(* IEC 61131-3 sources: elnaProjects/ElpcLogic/PomarKc7Changed/build_USO_ecl/_ (part 9) *)

FUNCTION nsCepeiControl : BOOL
  VAR_INPUT
    im : ImConfig;
  END_VAR

  nsCepeiControl:= NOT (
  	im.kran1.reliability OR
  	im.kran2.reliability OR
  	im.kran4.reliability OR
  	im.kran5.reliability OR
  	im.kran6.reliability OR
  	im.kran3b.reliability OR
  	im.pns.reliability OR
  	im.nu1.reliability OR
  	im.nu2.reliability OR
  	im.PNS.reliability OR
            im.v1_Avom.reliability OR
            im.v2_Avom.reliability OR
            (*im.Ten.reliability OR*)
  	im.mv.reliability);
END_FUNCTION

FUNCTION NapryageniaOK : BOOL
  VAR_INPUT
    im : ImConfig;
  END_VAR

  NapryageniaOK:=
  NOT (Im.SingleSignals.NS_G1_G2.Q
  OR Im.SingleSignals.NS_G10_G11.Q
  OR Im.SingleSignals.NS_G13_G14.Q
  OR Im.SingleSignals.NS_G15_G16.Q
  OR Im.SingleSignals.NS_G17.Q
  OR Im.SingleSignals.NS_G18_G19.Q
  OR Im.SingleSignals.NS_G3_G4.Q
  OR Im.SingleSignals.NS_G5_G6.Q
  OR Im.SingleSignals.NS_G7_G8.Q
  OR im.SingleSignals.QF1_on.Q
  OR Im.SingleSignals.QF2_on.Q
  OR Im.SingleSignals.QF23_on.Q
  OR Im.SingleSignals.QF4_QF5_on.Q
  OR Im.SingleSignals.QF6_QF7_on.Q
  OR Im.SingleSignals.QF8_QF9_on.Q
  OR Im.SingleSignals.QF10_QF11_on.Q
  OR im.SingleSignals.QF12_QF13_on.Q
  OR im.SingleSignals.QF22_on.Q
  OR Im.SingleSignals.QF14_QF15_on.Q);
END_FUNCTION

FUNCTION discretNS : BOOL
  VAR_INPUT
    di : DiConfig;
  END_VAR

  discretNS:=  ((di.di_0.reliability <> 255)
                OR (di.di_1.reliability <> 255)
                OR (di.di_2.reliability <> 255)
                OR (di.di_3.reliability <> 255)
                OR (di.di_4.reliability <> 255)
                OR (di.di_5.reliability <> 255)
                OR (di.di_6.reliability <> 255)
                OR (di.di_7.reliability <> 255)
                OR (di.di_8.reliability <> 255)
                OR (di.di_9.reliability <> 255)
                OR (di.di_10.reliability <> 255)
                OR (di.di_11.reliability <> 255)
                OR (di.di_12.reliability <> 255)
                OR (di.di_13.reliability <> 255)
                OR (di.di_14.reliability <> 255));
               (* OR (di.di_15.reliability <> 255)); *)
END_FUNCTION

FUNCTION BlockAllProtections : BOOL
  VAR_IN_OUT
    protections : ProtectionsConfig;
  END_VAR

  protections.Topornogo_podshipnika_EDT_1.inOpcCommandsDisabled:=TRUE;
  protections.Toy_podshipnika_EDT_2.inOpcCommandsDisabled:=TRUE;
  protections.Toy_podshipnika_kol_EDT_3.inOpcCommandsDisabled:=TRUE;
  protections.Toy_podshipnika_kol_EDT_4.inOpcCommandsDisabled:=TRUE;
  protections.To_podshipnika_shest_red_EDT_5.inOpcCommandsDisabled:=TRUE;
  protections.To_podshipnika_shest_red_EDT_6.inOpcCommandsDisabled:=TRUE;
  protections.To_podshipnika_N_EDT_7.inOpcCommandsDisabled:=TRUE;
  protections.To_podshipnika_svob_konca_EDT_8.inOpcCommandsDisabled:=TRUE;
  protections.Ty_podshipnika_rab_kol_EDT_9.inOpcCommandsDisabled:=TRUE;
  protections.Typornogo_podshipnika_nerab_kolodok_HT_10.inOpcCommandsDisabled:=TRUE;
  protections.Tgaza_na_vyhode_H.inOpcCommandsDisabled:=TRUE;
  protections.Os_sdvig_nagnetatelja_plus.inOpcCommandsDisabled:=TRUE;
  protections.Os_sdvig_nagnetatelja_minus.inOpcCommandsDisabled:=TRUE;
  protections.Pgaza_na_vyhode_nagnetatelia_GPA_STOP.inOpcCommandsDisabled:=TRUE;
  protections.Pgaza_na_vhode_nagnetatelia_GPA_STOP.inOpcCommandsDisabled:=TRUE;
  protections.Pgaza_na_vyhode_nagnetatelia.inOpcCommandsDisabled:=TRUE;
  protections.dPmaslo_gaz.inOpcCommandsDisabled:=TRUE;
  protections.Pmaslo_sm_nizkoe.inOpcCommandsDisabled:=TRUE;
  protections.Pmaslo_sm_vysokoe.inOpcCommandsDisabled:=TRUE;
  protections.Vibro_skorost_OPED_T1.inOpcCommandsDisabled:=TRUE;
  protections.Vibro_skorost_OPED_T2.inOpcCommandsDisabled:=TRUE;
  protections.Vibro_skorost_OYP_kolesa_ED_T3.inOpcCommandsDisabled:=TRUE;
  protections.Vibro_skorost_OP_kolesa_RH_T4.inOpcCommandsDisabled:=TRUE;
  protections.Vibro_skorost_OP_shesterni_RED_T5.inOpcCommandsDisabled:=TRUE;
  protections.Vibro_skorost_OP_shesterni_RED_T6.inOpcCommandsDisabled:=TRUE;
  protections.dPmaslo_gaz_less100.inOpcCommandsDisabled:=TRUE;
  protections.Reg_vozb_off.inOpcCommandsDisabled:=TRUE;
  protections.Fail_chastotnii_pusk.inOpcCommandsDisabled:=TRUE;
  protections.Off_avar_vikluchatel.inOpcCommandsDisabled:=TRUE;
  protections.AOKC_SHKC.inOpcCommandsDisabled:=TRUE;
  protections.AO_PRU.inOpcCommandsDisabled:=TRUE;
  protections.AO_ot_SHU.inOpcCommandsDisabled:=TRUE;
  protections.mvOff.inOpcCommandsDisabled:=TRUE;
  protections.Kran1_sdvig.inOpcCommandsDisabled:=TRUE;
  protections.Kran2_sdvig.inOpcCommandsDisabled:=TRUE;
END_FUNCTION

PROGRAM program0
  VAR
    SysTime : LREAL;
    systime_ns : ULINT;
    systime_s : ULINT;
    preSysTime : LREAL;
    tmpCycle : LREAL;
    preSys_s : ULINT;
    preSys_ns : ULINT;
  END_VAR
  VAR_EXTERNAL
    cur_Cycle : REAL;
    gStart_Tmr : REAL;
  END_VAR
  VAR
    Timings : fb_Timings;
    _init : BOOL      := TRUE;
    life_count : UINT;
    AI_structs_ini : proc_AI_Init;
    AI_Proc : proc_AI;
    AO_structs_ini : proc_AO_Init;
    AO_Proc : proc_AO;
    DI_structs_ini : proc_DI_Init;
    DI_Proc : proc_DI;
    DO_structs_ini : proc_DO_Init;
    DO_Proc : proc_DO;
    Get_algoritms_OPC : OPC_algoritms_set;
    Set_algoritms_OPC : OPC_algoritms_get;
    IM_structs_ini : proc_IM_Init;
    IM_Proc : proc_IM;
    Protections_structs_ini : proc_Protections_Init;
    Protections_Proc : proc_Protection;
    Algoritms_Proc : proc_algoritms;
    AlgoritmsManager : fb_AlgoritmsManager;
    ProtectionsManager : fb_ProtectionsManager;
  END_VAR
  VAR_EXTERNAL
    algManager : struct_AlgoritmsManager;
    protectManager : struct_ProtectionsManager;
  END_VAR

  (* Обработка времени. *)
  SysTime := ULINT_TO_LREAL(systime_s) + (1.0E-9 * ULINT_TO_LREAL(systime_ns));
  preSysTime := SysTime;
  tmpCycle := ULINT_TO_LREAL(systime_s - preSys_s) + 1.0E-9 * (ULINT_TO_LREAL(systime_ns) - ULINT_TO_LREAL(preSys_ns));
  cur_Cycle := LREAL_TO_REAL(tmpCycle);
  preSys_s := systime_s;
  preSys_ns := systime_ns;
  IF gStart_Tmr < 99999.9 THEN gStart_Tmr := gStart_Tmr + cur_Cycle; END_IF;
  Timings();

  IF  _init (*or external_init_ai *) then           (* Требуется инициализация структур и ФБ. *)
    (* Инициализация аналоговых входов. *)
      AI_structs_ini(init := TRUE);
      AI_Proc((*init := FALSE*));

    (* Инициализация дискретных входов. *)
      DI_structs_ini(init := TRUE);
      DI_Proc((*init := FALSE*));

      (* Инициализация аналоговых выходов. *)
  (*     AO_structs_ini(init := TRUE);
         AO_Proc(init := TRUE);*)

    (* Инициализация дискретных выходов. *)
      DO_structs_ini(init := TRUE);
      DO_Proc((*init := FALSE*));

     (* Инициализация ИМ. *)
      IM_structs_ini(init := TRUE);
      IM_Proc();

     (* Инициализация Защит *)
      Protections_structs_ini(init := TRUE);
      (*Protections_Proc();*)

       (* Стартовая инициализация OPC-тэгов элементами канальных структур. *)
          (*___________________AI______________________________________________________________________________*)
      (*ini_AI_OPC();*)

      _init := FALSE;

    ELSE                         (* Завершена инициализация структур и ФБ. *)

  (* Перенос OPC-тэгов в элементы структур каналов. *)
        (*___________________________________________AI________________________________________________*)
      (*Get_AI_OPC(); *)
       Get_algoritms_OPC();

     (* Пересчёт защит САУ. *)
     ProtectionsManager(protectManager);

       (* Пересчёт алгоритмов САУ. *)
     AlgoritmsManager(algManager);

      (****               Опрос входов.              ****)
          (* Опрос аналоговых входов. *)
      AI_Proc((*init := FALSE*));

          (* Опрос дискретных входов. *)
      DI_Proc((*init := FALSE*));

      (****              Запись выходов.             ****)
          (* Запись аналоговых выходов. *)
  (*    AO_Proc(init := FALSE);*)

       (* Запись дискретных выходов. *)
      DO_Proc((*init := FALSE*));

      (****               Опрос ИМ              ****)
      IM_Proc();

      (****            Опрос Защит              ****)
      Protections_Proc();

      Algoritms_Proc();

  END_IF;

  (* Передача информации на верхний уровень по OPC UA протоколу. *)
    (* Передача состояний каналов AI. *)
  (*Set_AI_OPC();)*
  (* Передача состояний каналов ИМ. *)
  (* Передача состояний защит. *)
  (* Передача состояний алгоритмов. *)
  Set_algoritms_OPC();
END_PROGRAM

CONFIGURATION config1
  VAR_GLOBAL
    systime_s AT %IL0.10.10 : ULINT;
    systime_ns AT %IL0.10.11 : ULINT;
    current_retrieve_us AT %IL0.10.12 : ULINT;
    current_config_us AT %IL0.10.13 : ULINT;
    current_publish_us AT %IL0.10.14 : ULINT;
    current_run_us AT %IL0.10.15 : ULINT;
    max_retrieve_us AT %QL0.10.16 : ULINT;
    max_config_us AT %QL0.10.17 : ULINT;
    max_publish_us AT %QL0.10.18 : ULINT;
    plc_run_number AT %IL0.10.19 : ULINT;
    arAIN_0 : TItemAIN;
    arAIN_1 : TItemAIN;
    arAIN_2 : TItemAIN;
    arAIN_3 : TItemAIN;
    arAIN_4 : TItemAIN;
    arAIN_5 : TItemAIN;
    arAIN_6 : TItemAIN;
    arAIN_7 : TItemAIN;
    arAIN_8 : TItemAIN;
    arAIN_9 : TItemAIN;
    arAIN_10 : TItemAIN;
    arAIN_11 : TItemAIN;
    arAIN_12 : TItemAIN;
    arAIN_13 : TItemAIN;
    arAIN_14 : TItemAIN;
    arAIN_15 : TItemAIN;
    arAIN_16 : TItemAIN;
    arAIN_17 : TItemAIN;
    arAIN_18 : TItemAIN;
    arAIN_19 : TItemAIN;
    arAIN_20 : TItemAIN;
    arAIN_21 : TItemAIN;
    arAIN_22 : TItemAIN;
    arAIN_23 : TItemAIN;
    arAIN_24 : TItemAIN;
    arAIN_25 : TItemAIN;
    arAIN_26 : TItemAIN;
    arAIN_27 : TItemAIN;
    arAIN_28 : TItemAIN;
    arAIN_29 : TItemAIN;
    arAIN_30 : TItemAIN;
    arAIN_31 : TItemAIN;
    arAIN_32 : TItemAIN;
    arAIN_33 : TItemAIN;
    arAIN_34 : TItemAIN;
    arAIN_35 : TItemAIN;
    arAIN_36 : TItemAIN;
    arAIN_37 : TItemAIN;
    arAIN_38 : TItemAIN;
    arAIN_39 : TItemAIN;
    arAIN_40 : TItemAIN;
    arAIN_41 : TItemAIN;
    arAIN_42 : TItemAIN;
    arAIN_43 : TItemAIN;
    arAIN_44 : TItemAIN;
    arAIN_45 : TItemAIN;
    arAIN_46 : TItemAIN;
    arAIN_47 : TItemAIN;
    arAIN_48 : TItemAIN;
    arAIN_49 : TItemAIN;
    arAIN_50 : TItemAIN;
    arAIN_51 : TItemAIN;
    arAIN_52 : TItemAIN;
    arAIN_53 : TItemAIN;
    arAIN_54 : TItemAIN;
    arAIN_55 : TItemAIN;
    arAIN_56 : TItemAIN;
    arAIN_57 : TItemAIN;
    arAIN_58 : TItemAIN;
    arAIN_59 : TItemAIN;
    arAIN_60 : TItemAIN;
    arAIN_61 : TItemAIN;
    arAIN_62 : TItemAIN;
    arAIN_63 : TItemAIN;
    arAIN_64 : TItemAIN;
    arAIN_65 : TItemAIN;
    arAIN_66 : TItemAIN;
    arAIN_67 : TItemAIN;
    arAIN_68 : TItemAIN;
    arAIN_69 : TItemAIN;
    arAIN_70 : TItemAIN;
    arAIN_71 : TItemAIN;
    arAIN_72 : TItemAIN;
    arAIN_73 : TItemAIN;
    arAIN_74 : TItemAIN;
    arAIN_75 : TItemAIN;
    arAIN_76 : TItemAIN;
    arAIN_77 : TItemAIN;
    arAIN_78 : TItemAIN;
    arAIN_79 : TItemAIN;
    arDIN_0 : TItemDIN;
    arDIN_1 : TItemDIN;
    arDIN_2 : TItemDIN;
    arDIN_3 : TItemDIN;
    arDIN_4 : TItemDIN;
    arDIN_5 : TItemDIN;
    arDIN_6 : TItemDIN;
    arDIN_7 : TItemDIN;
    arDIN_8 : TItemDIN;
    arDIN_9 : TItemDIN;
    arDIN_10 : TItemDIN;
    arDIN_11 : TItemDIN;
    arDIN_12 : TItemDIN;
    arDIN_13 : TItemDIN;
    arDIN_14 : TItemDIN;
    arDIN_15 : TItemDIN;
    arDIN_16 : TItemDIN;
    arDIN_17 : TItemDIN;
    arDIN_18 : TItemDIN;
    arDIN_19 : TItemDIN;
    arDIN_20 : TItemDIN;
    arDIN_21 : TItemDIN;
    arAOUT_0 : TDoubleData;
    arAOUT_1 : TDoubleData;
    arDOUT_0 : TWordData;
    arDOUT_1 : TWordData;
    arDOUT_2 : TWordData;
    arDOUT_3 : TWordData;
    arDOUT_4 : TWordData;
    arDOUT_66 : TWordData;
    arERR_0 : TItemDIN;
    arERR_1 : TItemDIN;
    arERR_2 : TItemDIN;
    arERR_3 : TItemDIN;
    arERR_4 : TItemDIN;
    arERR_5 : TItemDIN;
    arERR_6 : TItemDIN;
    arERR_7 : TItemDIN;
    arERR_8 : TItemDIN;
    arERR_9 : TItemDIN;
    arERR_10 : TItemDIN;
    arERR_11 : TItemDIN;
    arERR_12 : TItemDIN;
    arERR_13 : TItemDIN;
    arERR_14 : TItemDIN;
    arERR_15 : TItemDIN;
    arERR_16 : TItemDIN;
    arERR_17 : TItemDIN;
    arERR_18 : TItemDIN;
    arERR_19 : TItemDIN;
    arERR_20 : TItemDIN;
    arERR_21 : TItemDIN;
    arERR_22 : TItemDIN;
    arERR_23 : TItemDIN;
    arERR_24 : TItemDIN;
    arERR_66 : TItemDIN;
    arRelSt_0 : TItemDIN;
  END_VAR

  RESOURCE resource1 ON PLC
    VAR_GLOBAL CONSTANT
      gMaint_Time : REAL;
    END_VAR
    VAR_GLOBAL
      cur_Cycle : REAL;
      gStart_Tmr : REAL;
    END_VAR
    VAR_GLOBAL CONSTANT
      req_Cycle : REAL := 0.02;
    END_VAR
    VAR_GLOBAL
      gF_T_100mSec : BOOL;
      gT_1Sec : BOOL;
      gF_T_1Sec : BOOL;
      gT_1Min : BOOL;
      gR_T_1Min : BOOL;
      gF_T_1Min : BOOL;
      T_1SEC : REAL;
      del_T : REAL;
      ai : AiConfig;
      di : DiConfig;
      od : DOconfig;
      ao : AOConfig;
      IM : ImConfig;
      protections : ProtectionsConfig;
      algoritms : AlgoritmsConfig;
      algManager : struct_AlgoritmsManager;
      ModeGpa : TYPE_ModeGpa;
      protectManager : struct_ProtectionsManager;
      NotHasRezervNU : BOOL;
      Reset_HasNU : BOOL;
      AlgTimers : struct_AlgTimers;
      AlgQuestions : AlgoritmsQuestions;
      PMcommand : TYPE_CommandsPotectionsManager;
      AI_Aktivnaia_moshchnost_HL AT %QL0.2 : LREAL;
      AI_Aktivnaia_moshchnost_LL AT %QL0.3 : LREAL;
      AI_Aktivnaia_moshchnost_command AT %QW0.1 : UINT;
      AI_Aktivnaia_moshchnost_newHL AT %QL0.4 : LREAL;
      AI_Aktivnaia_moshchnost_newLL AT %QL0.5 : LREAL;
      AI_Aktivnaia_moshchnost_status AT %QD0.6 : UDINT;
      AI_Aktivnaia_moshchnost_value AT %QL0.7 : LREAL;
      AI_Osevoi_sdvig_rotora_nagnetatelia_HA AT %QL0.27 : LREAL;
      AI_Osevoi_sdvig_rotora_nagnetatelia_HL AT %QL0.28 : LREAL;
      AI_Osevoi_sdvig_rotora_nagnetatelia_HW AT %QL0.29 : LREAL;
      AI_Osevoi_sdvig_rotora_nagnetatelia_LA AT %QL0.30 : LREAL;
      AI_Osevoi_sdvig_rotora_nagnetatelia_LL AT %QL0.31 : LREAL;
      AI_Osevoi_sdvig_rotora_nagnetatelia_LW AT %QL0.32 : LREAL;
      AI_Osevoi_sdvig_rotora_nagnetatelia_command AT %QW0.26 : UINT;
      AI_Osevoi_sdvig_rotora_nagnetatelia_newHA AT %QL0.33 : LREAL;
      AI_Osevoi_sdvig_rotora_nagnetatelia_newHL AT %QL0.34 : LREAL;
      AI_Osevoi_sdvig_rotora_nagnetatelia_newHW AT %QL0.35 : LREAL;
      AI_Osevoi_sdvig_rotora_nagnetatelia_newLA AT %QL0.36 : LREAL;
      AI_Osevoi_sdvig_rotora_nagnetatelia_newLL AT %QL0.37 : LREAL;
      AI_Osevoi_sdvig_rotora_nagnetatelia_newLW AT %QL0.38 : LREAL;
      AI_Osevoi_sdvig_rotora_nagnetatelia_status AT %QD0.39 : UDINT;
      AI_Osevoi_sdvig_rotora_nagnetatelia_value AT %QL0.40 : LREAL;
      AI_P_gaza_na_vkhode_nagnetatelia_HL AT %QL0.42 : LREAL;
      AI_P_gaza_na_vkhode_nagnetatelia_LL AT %QL0.43 : LREAL;
      AI_P_gaza_na_vkhode_nagnetatelia_command AT %QW0.41 : UINT;
      AI_P_gaza_na_vkhode_nagnetatelia_newHL AT %QL0.44 : LREAL;
      AI_P_gaza_na_vkhode_nagnetatelia_newLL AT %QL0.45 : LREAL;
      AI_P_gaza_na_vkhode_nagnetatelia_status AT %QD0.46 : UDINT;
      AI_P_gaza_na_vkhode_nagnetatelia_value AT %QL0.47 : LREAL;
      AI_P_gaza_na_vykhode_nagnetatelia_HL AT %QL0.49 : LREAL;
      AI_P_gaza_na_vykhode_nagnetatelia_LL AT %QL0.50 : LREAL;
      AI_P_gaza_na_vykhode_nagnetatelia_command AT %QW0.48 : UINT;
      AI_P_gaza_na_vykhode_nagnetatelia_newHL AT %QL0.51 : LREAL;
      AI_P_gaza_na_vykhode_nagnetatelia_newLL AT %QL0.52 : LREAL;
      AI_P_gaza_na_vykhode_nagnetatelia_status AT %QD0.53 : UDINT;
      AI_P_gaza_na_vykhode_nagnetatelia_value AT %QL0.54 : LREAL;
      AI_P_masla_smazki_nizkoe_HL AT %QL0.56 : LREAL;
      AI_P_masla_smazki_nizkoe_LA AT %QL0.57 : LREAL;
      AI_P_masla_smazki_nizkoe_LL AT %QL0.58 : LREAL;
      AI_P_masla_smazki_nizkoe_LW AT %QL0.59 : LREAL;
      AI_P_masla_smazki_nizkoe_command AT %QW0.55 : UINT;
      AI_P_masla_smazki_nizkoe_newHL AT %QL0.60 : LREAL;
      AI_P_masla_smazki_nizkoe_newLA AT %QL0.61 : LREAL;
      AI_P_masla_smazki_nizkoe_newLL AT %QL0.62 : LREAL;
      AI_P_masla_smazki_nizkoe_newLW AT %QL0.63 : LREAL;
      AI_P_masla_smazki_nizkoe_status AT %QD0.64 : UDINT;
      AI_P_masla_smazki_nizkoe_value AT %QL0.65 : LREAL;
      AI_P_masla_smazki_srednee_posle_nasosov_HL AT %QL0.67 : LREAL;
      AI_P_masla_smazki_srednee_posle_nasosov_LL AT %QL0.68 : LREAL;
      AI_P_masla_smazki_srednee_posle_nasosov_LW AT %QL0.69 : LREAL;
      AI_P_masla_smazki_srednee_posle_nasosov_command AT %QW0.66 : UINT;
      AI_P_masla_smazki_srednee_posle_nasosov_newHL AT %QL0.70 : LREAL;
      AI_P_masla_smazki_srednee_posle_nasosov_newLL AT %QL0.71 : LREAL;
      AI_P_masla_smazki_srednee_posle_nasosov_newLW AT %QL0.72 : LREAL;
      AI_P_masla_smazki_srednee_posle_nasosov_status AT %QD0.73 : UDINT;
      AI_P_masla_smazki_srednee_posle_nasosov_value AT %QL0.74 : LREAL;
      AI_P_masla_uplotneniia_HL AT %QL0.76 : LREAL;
      AI_P_masla_uplotneniia_LL AT %QL0.77 : LREAL;
      AI_P_masla_uplotneniia_command AT %QW0.75 : UINT;
      AI_P_masla_uplotneniia_newHL AT %QL0.78 : LREAL;
      AI_P_masla_uplotneniia_newLL AT %QL0.79 : LREAL;
      AI_P_masla_uplotneniia_status AT %QD0.80 : UDINT;
      AI_P_masla_uplotneniia_value AT %QL0.81 : LREAL;
      AI_Reaktivnaia_moshchnost_HL AT %QL0.83 : LREAL;
      AI_Reaktivnaia_moshchnost_LL AT %QL0.84 : LREAL;
      AI_Reaktivnaia_moshchnost_command AT %QW0.82 : UINT;
      AI_Reaktivnaia_moshchnost_newHL AT %QL0.85 : LREAL;
      AI_Reaktivnaia_moshchnost_newLL AT %QL0.86 : LREAL;
      AI_Reaktivnaia_moshchnost_status AT %QD0.87 : UDINT;
      AI_Reaktivnaia_moshchnost_value AT %QL0.88 : LREAL;
      AI_T_aktivnogo_zheleza_statora_1_k_HL AT %QL0.90 : LREAL;
      AI_T_aktivnogo_zheleza_statora_1_k_LL AT %QL0.91 : LREAL;
      AI_T_aktivnogo_zheleza_statora_1_k_command AT %QW0.89 : UINT;
      AI_T_aktivnogo_zheleza_statora_1_k_newHL AT %QL0.92 : LREAL;
      AI_T_aktivnogo_zheleza_statora_1_k_newLL AT %QL0.93 : LREAL;
      AI_T_aktivnogo_zheleza_statora_1_k_status AT %QD0.94 : UDINT;
      AI_T_aktivnogo_zheleza_statora_1_k_value AT %QL0.95 : LREAL;
      AI_T_aktivnogo_zheleza_statora_2_k_HL AT %QL0.97 : LREAL;
      AI_T_aktivnogo_zheleza_statora_2_k_LL AT %QL0.98 : LREAL;
      AI_T_aktivnogo_zheleza_statora_2_k_command AT %QW0.96 : UINT;
      AI_T_aktivnogo_zheleza_statora_2_k_newHL AT %QL0.99 : LREAL;
      AI_T_aktivnogo_zheleza_statora_2_k_newLL AT %QL0.100 : LREAL;
      AI_T_aktivnogo_zheleza_statora_2_k_status AT %QD0.101 : UDINT;
      AI_T_aktivnogo_zheleza_statora_2_k_value AT %QL0.102 : LREAL;
      AI_T_aktivnogo_zheleza_statora_3_k_HL AT %QL0.104 : LREAL;
      AI_T_aktivnogo_zheleza_statora_3_k_LL AT %QL0.105 : LREAL;
      AI_T_aktivnogo_zheleza_statora_3_k_command AT %QW0.103 : UINT;
      AI_T_aktivnogo_zheleza_statora_3_k_newHL AT %QL0.106 : LREAL;
      AI_T_aktivnogo_zheleza_statora_3_k_newLL AT %QL0.107 : LREAL;
      AI_T_aktivnogo_zheleza_statora_3_k_status AT %QD0.108 : UDINT;
      AI_T_aktivnogo_zheleza_statora_3_k_value AT %QL0.109 : LREAL;
      AI_T_clodAir_dvigatelia_t1_HL AT %QL0.111 : LREAL;
      AI_T_clodAir_dvigatelia_t1_LL AT %QL0.112 : LREAL;
      AI_T_clodAir_dvigatelia_t1_command AT %QW0.110 : UINT;
      AI_T_clodAir_dvigatelia_t1_newHL AT %QL0.113 : LREAL;
      AI_T_clodAir_dvigatelia_t1_newLL AT %QL0.114 : LREAL;
      AI_T_clodAir_dvigatelia_t1_status AT %QD0.115 : UDINT;
      AI_T_clodAir_dvigatelia_t1_value AT %QL0.116 : LREAL;
      AI_T_gaz_in_nagnetatelia_HL AT %QL0.118 : LREAL;
      AI_T_gaz_in_nagnetatelia_LL AT %QL0.119 : LREAL;
      AI_T_gaz_in_nagnetatelia_command AT %QW0.117 : UINT;
      AI_T_gaz_in_nagnetatelia_newHL AT %QL0.120 : LREAL;
      AI_T_gaz_in_nagnetatelia_newLL AT %QL0.121 : LREAL;
      AI_T_gaz_in_nagnetatelia_status AT %QD0.122 : UDINT;
      AI_T_gaz_in_nagnetatelia_value AT %QL0.123 : LREAL;
      AI_T_gaz_out_nagnetatelia_HA AT %QL0.125 : LREAL;
      AI_T_gaz_out_nagnetatelia_HL AT %QL0.126 : LREAL;
      AI_T_gaz_out_nagnetatelia_HW AT %QL0.127 : LREAL;
      AI_T_gaz_out_nagnetatelia_LL AT %QL0.128 : LREAL;
      AI_T_gaz_out_nagnetatelia_command AT %QW0.124 : UINT;
      AI_T_gaz_out_nagnetatelia_newHA AT %QL0.129 : LREAL;
      AI_T_gaz_out_nagnetatelia_newHL AT %QL0.130 : LREAL;
      AI_T_gaz_out_nagnetatelia_newHW AT %QL0.131 : LREAL;
      AI_T_gaz_out_nagnetatelia_newLL AT %QL0.132 : LREAL;
      AI_T_gaz_out_nagnetatelia_status AT %QD0.133 : UDINT;
      AI_T_gaz_out_nagnetatelia_value AT %QL0.134 : LREAL;
      AI_T_hotAir_dvigatelia_t1_HL AT %QL0.136 : LREAL;
      AI_T_hotAir_dvigatelia_t1_LL AT %QL0.137 : LREAL;
      AI_T_hotAir_dvigatelia_t1_command AT %QW0.135 : UINT;
      AI_T_hotAir_dvigatelia_t1_newHL AT %QL0.138 : LREAL;
      AI_T_hotAir_dvigatelia_t1_newLL AT %QL0.139 : LREAL;
      AI_T_hotAir_dvigatelia_t1_status AT %QD0.140 : UDINT;
      AI_T_hotAir_dvigatelia_t1_value AT %QL0.141 : LREAL;
      AI_T_masla_do_AVOM_HL AT %QL0.143 : LREAL;
      AI_T_masla_do_AVOM_LL AT %QL0.144 : LREAL;
      AI_T_masla_do_AVOM_command AT %QW0.142 : UINT;
      AI_T_masla_do_AVOM_newHL AT %QL0.145 : LREAL;
      AI_T_masla_do_AVOM_newLL AT %QL0.146 : LREAL;
      AI_T_masla_do_AVOM_status AT %QD0.147 : UDINT;
      AI_T_masla_do_AVOM_value AT %QL0.148 : LREAL;
      AI_T_masla_na_slive_perednego_opornogo_podshipnika_dvigatelia_HL AT %QL0.150 : LREAL;
      AI_T_masla_na_slive_perednego_opornogo_podshipnika_dvigatelia_LL AT %QL0.151 : LREAL;
      AI_T_masla_na_slive_perednego_opornogo_podshipnika_dvigatelia_command AT %QW0.149 : UINT;
      AI_T_masla_na_slive_perednego_opornogo_podshipnika_dvigatelia_newHL AT %QL0.152 : LREAL;
      AI_T_masla_na_slive_perednego_opornogo_podshipnika_dvigatelia_newLL AT %QL0.153 : LREAL;
      AI_T_masla_na_slive_perednego_opornogo_podshipnika_dvigatelia_status AT %QD0.154 : UDINT;
      AI_T_masla_na_slive_perednego_opornogo_podshipnika_dvigatelia_value AT %QL0.155 : LREAL;
      AI_T_masla_na_slive_zadnego_opornogo_podshipnika_dvigatelia_HL AT %QL0.157 : LREAL;
      AI_T_masla_na_slive_zadnego_opornogo_podshipnika_dvigatelia_LL AT %QL0.158 : LREAL;
      AI_T_masla_na_slive_zadnego_opornogo_podshipnika_dvigatelia_command AT %QW0.156 : UINT;
      AI_T_masla_na_slive_zadnego_opornogo_podshipnika_dvigatelia_newHL AT %QL0.159 : LREAL;
      AI_T_masla_na_slive_zadnego_opornogo_podshipnika_dvigatelia_newLL AT %QL0.160 : LREAL;
      AI_T_masla_na_slive_zadnego_opornogo_podshipnika_dvigatelia_status AT %QD0.161 : UDINT;
      AI_T_masla_na_slive_zadnego_opornogo_podshipnika_dvigatelia_value AT %QL0.162 : LREAL;
      AI_T_masla_posle_AVOM_HL AT %QL0.164 : LREAL;
      AI_T_masla_posle_AVOM_LL AT %QL0.165 : LREAL;
      AI_T_masla_posle_AVOM_command AT %QW0.163 : UINT;
      AI_T_masla_posle_AVOM_newHL AT %QL0.166 : LREAL;
      AI_T_masla_posle_AVOM_newLL AT %QL0.167 : LREAL;
      AI_T_masla_posle_AVOM_status AT %QD0.168 : UDINT;
      AI_T_masla_posle_AVOM_value AT %QL0.169 : LREAL;
      AI_T_masla_v_maslobake_HL AT %QL0.171 : LREAL;
      AI_T_masla_v_maslobake_HW AT %QL0.172 : LREAL;
      AI_T_masla_v_maslobake_LL AT %QL0.173 : LREAL;
      AI_T_masla_v_maslobake_LW AT %QL0.174 : LREAL;
      AI_T_masla_v_maslobake_command AT %QW0.170 : UINT;
      AI_T_masla_v_maslobake_newHL AT %QL0.175 : LREAL;
      AI_T_masla_v_maslobake_newHW AT %QL0.176 : LREAL;
      AI_T_masla_v_maslobake_newLL AT %QL0.177 : LREAL;
      AI_T_masla_v_maslobake_newLW AT %QL0.178 : LREAL;
      AI_T_masla_v_maslobake_status AT %QD0.179 : UDINT;
      AI_T_masla_v_maslobake_value AT %QL0.180 : LREAL;
      AI_T_obmotki_fazy_1_k_HL AT %QL0.182 : LREAL;
      AI_T_obmotki_fazy_1_k_LL AT %QL0.183 : LREAL;
      AI_T_obmotki_fazy_1_k_command AT %QW0.181 : UINT;
      AI_T_obmotki_fazy_1_k_newHL AT %QL0.184 : LREAL;
      AI_T_obmotki_fazy_1_k_newLL AT %QL0.185 : LREAL;
      AI_T_obmotki_fazy_1_k_status AT %QD0.186 : UDINT;
      AI_T_obmotki_fazy_1_k_value AT %QL0.187 : LREAL;
      AI_T_obmotki_fazy_2_k_HL AT %QL0.189 : LREAL;
      AI_T_obmotki_fazy_2_k_LL AT %QL0.190 : LREAL;
      AI_T_obmotki_fazy_2_k_command AT %QW0.188 : UINT;
      AI_T_obmotki_fazy_2_k_newHL AT %QL0.191 : LREAL;
      AI_T_obmotki_fazy_2_k_newLL AT %QL0.192 : LREAL;
      AI_T_obmotki_fazy_2_k_status AT %QD0.193 : UDINT;
      AI_T_obmotki_fazy_2_k_value AT %QL0.194 : LREAL;
      AI_T_obmotki_fazy_3_k_HL AT %QL0.196 : LREAL;
      AI_T_obmotki_fazy_3_k_LL AT %QL0.197 : LREAL;
      AI_T_obmotki_fazy_3_k_command AT %QW0.195 : UINT;
      AI_T_obmotki_fazy_3_k_newHL AT %QL0.198 : LREAL;
      AI_T_obmotki_fazy_3_k_newLL AT %QL0.199 : LREAL;
      AI_T_obmotki_fazy_3_k_status AT %QD0.200 : UDINT;
      AI_T_obmotki_fazy_3_k_value AT %QL0.201 : LREAL;
      AI_T_oporno_upornogo_podshipnika_nagnetatelia_t4_HA AT %QL0.203 : LREAL;
      AI_T_oporno_upornogo_podshipnika_nagnetatelia_t4_HL AT %QL0.204 : LREAL;
      AI_T_oporno_upornogo_podshipnika_nagnetatelia_t4_HW AT %QL0.205 : LREAL;
      AI_T_oporno_upornogo_podshipnika_nagnetatelia_t4_LL AT %QL0.206 : LREAL;
      AI_T_oporno_upornogo_podshipnika_nagnetatelia_t4_command AT %QW0.202 : UINT;
      AI_T_oporno_upornogo_podshipnika_nagnetatelia_t4_newHA AT %QL0.207 : LREAL;
      AI_T_oporno_upornogo_podshipnika_nagnetatelia_t4_newHL AT %QL0.208 : LREAL;
      AI_T_oporno_upornogo_podshipnika_nagnetatelia_t4_newHW AT %QL0.209 : LREAL;
      AI_T_oporno_upornogo_podshipnika_nagnetatelia_t4_newLL AT %QL0.210 : LREAL;
      AI_T_oporno_upornogo_podshipnika_nagnetatelia_t4_status AT %QD0.211 : UDINT;
      AI_T_oporno_upornogo_podshipnika_nagnetatelia_t4_value AT %QL0.212 : LREAL;
      AI_T_opornogo_podshipnika_nagnetatelia_t1_HA AT %QL0.214 : LREAL;
      AI_T_opornogo_podshipnika_nagnetatelia_t1_HL AT %QL0.215 : LREAL;
      AI_T_opornogo_podshipnika_nagnetatelia_t1_HW AT %QL0.216 : LREAL;
      AI_T_opornogo_podshipnika_nagnetatelia_t1_LL AT %QL0.217 : LREAL;
      AI_T_opornogo_podshipnika_nagnetatelia_t1_command AT %QW0.213 : UINT;
      AI_T_opornogo_podshipnika_nagnetatelia_t1_newHA AT %QL0.218 : LREAL;
      AI_T_opornogo_podshipnika_nagnetatelia_t1_newHL AT %QL0.219 : LREAL;
      AI_T_opornogo_podshipnika_nagnetatelia_t1_newHW AT %QL0.220 : LREAL;
      AI_T_opornogo_podshipnika_nagnetatelia_t1_newLL AT %QL0.221 : LREAL;
      AI_T_opornogo_podshipnika_nagnetatelia_t1_status AT %QD0.222 : UDINT;
      AI_T_opornogo_podshipnika_nagnetatelia_t1_value AT %QL0.223 : LREAL;
      AI_T_opornogo_podshipnika_nagnetatelia_t2_HA AT %QL0.225 : LREAL;
      AI_T_opornogo_podshipnika_nagnetatelia_t2_HL AT %QL0.226 : LREAL;
      AI_T_opornogo_podshipnika_nagnetatelia_t2_HW AT %QL0.227 : LREAL;
      AI_T_opornogo_podshipnika_nagnetatelia_t2_LL AT %QL0.228 : LREAL;
      AI_T_opornogo_podshipnika_nagnetatelia_t2_command AT %QW0.224 : UINT;
      AI_T_opornogo_podshipnika_nagnetatelia_t2_newHA AT %QL0.229 : LREAL;
      AI_T_opornogo_podshipnika_nagnetatelia_t2_newHL AT %QL0.230 : LREAL;
      AI_T_opornogo_podshipnika_nagnetatelia_t2_newHW AT %QL0.231 : LREAL;
      AI_T_opornogo_podshipnika_nagnetatelia_t2_newLL AT %QL0.232 : LREAL;
      AI_T_opornogo_podshipnika_nagnetatelia_t2_status AT %QD0.233 : UDINT;
      AI_T_opornogo_podshipnika_nagnetatelia_t2_value AT %QL0.234 : LREAL;
      AI_T_opornogo_podshipnika_nagnetatelia_t3_HA AT %QL0.236 : LREAL;
      AI_T_opornogo_podshipnika_nagnetatelia_t3_HL AT %QL0.237 : LREAL;
      AI_T_opornogo_podshipnika_nagnetatelia_t3_HW AT %QL0.238 : LREAL;
      AI_T_opornogo_podshipnika_nagnetatelia_t3_LL AT %QL0.239 : LREAL;
      AI_T_opornogo_podshipnika_nagnetatelia_t3_command AT %QW0.235 : UINT;
      AI_T_opornogo_podshipnika_nagnetatelia_t3_newHA AT %QL0.240 : LREAL;
      AI_T_opornogo_podshipnika_nagnetatelia_t3_newHL AT %QL0.241 : LREAL;
      AI_T_opornogo_podshipnika_nagnetatelia_t3_newHW AT %QL0.242 : LREAL;
      AI_T_opornogo_podshipnika_nagnetatelia_t3_newLL AT %QL0.243 : LREAL;
      AI_T_opornogo_podshipnika_nagnetatelia_t3_status AT %QD0.244 : UDINT;
      AI_T_opornogo_podshipnika_nagnetatelia_t3_value AT %QL0.245 : LREAL;
      AI_T_perednego_opornogo_podshipnika_dvigatelia_t1_HA AT %QL0.247 : LREAL;
      AI_T_perednego_opornogo_podshipnika_dvigatelia_t1_HL AT %QL0.248 : LREAL;
      AI_T_perednego_opornogo_podshipnika_dvigatelia_t1_HW AT %QL0.249 : LREAL;
      AI_T_perednego_opornogo_podshipnika_dvigatelia_t1_LL AT %QL0.250 : LREAL;
      AI_T_perednego_opornogo_podshipnika_dvigatelia_t1_command AT %QW0.246 : UINT;
      AI_T_perednego_opornogo_podshipnika_dvigatelia_t1_newHA AT %QL0.251 : LREAL;
      AI_T_perednego_opornogo_podshipnika_dvigatelia_t1_newHL AT %QL0.252 : LREAL;
      AI_T_perednego_opornogo_podshipnika_dvigatelia_t1_newHW AT %QL0.253 : LREAL;
      AI_T_perednego_opornogo_podshipnika_dvigatelia_t1_newLL AT %QL0.254 : LREAL;
      AI_T_perednego_opornogo_podshipnika_dvigatelia_t1_status AT %QD0.255 : UDINT;
      AI_T_perednego_opornogo_podshipnika_dvigatelia_t1_value AT %QL0.256 : LREAL;
      AI_T_podshipnika_reduktora_t1_HA AT %QL0.258 : LREAL;
      AI_T_podshipnika_reduktora_t1_HL AT %QL0.259 : LREAL;
      AI_T_podshipnika_reduktora_t1_HW AT %QL0.260 : LREAL;
      AI_T_podshipnika_reduktora_t1_LL AT %QL0.261 : LREAL;
      AI_T_podshipnika_reduktora_t1_command AT %QW0.257 : UINT;
      AI_T_podshipnika_reduktora_t1_newHA AT %QL0.262 : LREAL;
      AI_T_podshipnika_reduktora_t1_newHL AT %QL0.263 : LREAL;
      AI_T_podshipnika_reduktora_t1_newHW AT %QL0.264 : LREAL;
      AI_T_podshipnika_reduktora_t1_newLL AT %QL0.265 : LREAL;
      AI_T_podshipnika_reduktora_t1_status AT %QD0.266 : UDINT;
      AI_T_podshipnika_reduktora_t1_value AT %QL0.267 : LREAL;
      AI_T_podshipnika_reduktora_t2_HA AT %QL0.269 : LREAL;
      AI_T_podshipnika_reduktora_t2_HL AT %QL0.270 : LREAL;
      AI_T_podshipnika_reduktora_t2_HW AT %QL0.271 : LREAL;
      AI_T_podshipnika_reduktora_t2_LL AT %QL0.272 : LREAL;
      AI_T_podshipnika_reduktora_t2_command AT %QW0.268 : UINT;
      AI_T_podshipnika_reduktora_t2_newHA AT %QL0.273 : LREAL;
      AI_T_podshipnika_reduktora_t2_newHL AT %QL0.274 : LREAL;
      AI_T_podshipnika_reduktora_t2_newHW AT %QL0.275 : LREAL;
      AI_T_podshipnika_reduktora_t2_newLL AT %QL0.276 : LREAL;
      AI_T_podshipnika_reduktora_t2_status AT %QD0.277 : UDINT;
      AI_T_podshipnika_reduktora_t2_value AT %QL0.278 : LREAL;
      AI_T_podshipnika_reduktora_t3_HA AT %QL0.280 : LREAL;
      AI_T_podshipnika_reduktora_t3_HL AT %QL0.281 : LREAL;
      AI_T_podshipnika_reduktora_t3_HW AT %QL0.282 : LREAL;
      AI_T_podshipnika_reduktora_t3_LL AT %QL0.283 : LREAL;
      AI_T_podshipnika_reduktora_t3_command AT %QW0.279 : UINT;
      AI_T_podshipnika_reduktora_t3_newHA AT %QL0.284 : LREAL;
      AI_T_podshipnika_reduktora_t3_newHL AT %QL0.285 : LREAL;
      AI_T_podshipnika_reduktora_t3_newHW AT %QL0.286 : LREAL;
      AI_T_podshipnika_reduktora_t3_newLL AT %QL0.287 : LREAL;
      AI_T_podshipnika_reduktora_t3_status AT %QD0.288 : UDINT;
      AI_T_podshipnika_reduktora_t3_value AT %QL0.289 : LREAL;
      AI_T_podshipnika_reduktora_t4_HA AT %QL0.291 : LREAL;
      AI_T_podshipnika_reduktora_t4_HL AT %QL0.292 : LREAL;
      AI_T_podshipnika_reduktora_t4_HW AT %QL0.293 : LREAL;
      AI_T_podshipnika_reduktora_t4_LL AT %QL0.294 : LREAL;
      AI_T_podshipnika_reduktora_t4_command AT %QW0.290 : UINT;
      AI_T_podshipnika_reduktora_t4_newHA AT %QL0.295 : LREAL;
      AI_T_podshipnika_reduktora_t4_newHL AT %QL0.296 : LREAL;
      AI_T_podshipnika_reduktora_t4_newHW AT %QL0.297 : LREAL;
      AI_T_podshipnika_reduktora_t4_newLL AT %QL0.298 : LREAL;
      AI_T_podshipnika_reduktora_t4_status AT %QD0.299 : UDINT;
      AI_T_podshipnika_reduktora_t4_value AT %QL0.300 : LREAL;
      AI_T_vnytri_shkafa_HL AT %QL0.866 : LREAL;
      AI_T_vnytri_shkafa_HW AT %QL0.870 : LREAL;
      AI_T_vnytri_shkafa_LL AT %QL0.867 : LREAL;
      AI_T_vnytri_shkafa_LW AT %QL0.872 : LREAL;
      AI_T_vnytri_shkafa_command AT %QW0.863 : UINT;
      AI_T_vnytri_shkafa_newHL AT %QL0.868 : LREAL;
      AI_T_vnytri_shkafa_newHW AT %QL0.871 : LREAL;
      AI_T_vnytri_shkafa_newLL AT %QL0.869 : LREAL;
      AI_T_vnytri_shkafa_newLW AT %QL0.873 : LREAL;
      AI_T_vnytri_shkafa_status AT %QD0.864 : UDINT;
      AI_T_vnytri_shkafa_value AT %QL0.865 : LREAL;
      AI_T_zadnego_opornogo_podshipnika_dvigatelia_t2_HA AT %QL0.302 : LREAL;
      AI_T_zadnego_opornogo_podshipnika_dvigatelia_t2_HL AT %QL0.303 : LREAL;
      AI_T_zadnego_opornogo_podshipnika_dvigatelia_t2_HW AT %QL0.304 : LREAL;
      AI_T_zadnego_opornogo_podshipnika_dvigatelia_t2_LL AT %QL0.305 : LREAL;
      AI_T_zadnego_opornogo_podshipnika_dvigatelia_t2_command AT %QW0.301 : UINT;
      AI_T_zadnego_opornogo_podshipnika_dvigatelia_t2_newHA AT %QL0.306 : LREAL;
      AI_T_zadnego_opornogo_podshipnika_dvigatelia_t2_newHL AT %QL0.307 : LREAL;
      AI_T_zadnego_opornogo_podshipnika_dvigatelia_t2_newHW AT %QL0.308 : LREAL;
      AI_T_zadnego_opornogo_podshipnika_dvigatelia_t2_newLL AT %QL0.309 : LREAL;
      AI_T_zadnego_opornogo_podshipnika_dvigatelia_t2_status AT %QD0.310 : UDINT;
      AI_T_zadnego_opornogo_podshipnika_dvigatelia_t2_value AT %QL0.311 : LREAL;
      AI_Tok_statora_elektrodvigatelia_HL AT %QL0.313 : LREAL;
      AI_Tok_statora_elektrodvigatelia_LL AT %QL0.314 : LREAL;
      AI_Tok_statora_elektrodvigatelia_command AT %QW0.312 : UINT;
      AI_Tok_statora_elektrodvigatelia_newHL AT %QL0.315 : LREAL;
      AI_Tok_statora_elektrodvigatelia_newLL AT %QL0.316 : LREAL;
      AI_Tok_statora_elektrodvigatelia_status AT %QD0.317 : UDINT;
      AI_Tok_statora_elektrodvigatelia_value AT %QL0.318 : LREAL;
      AI_Tok_vozbuzhdeniia_vozbuditelia_HL AT %QL0.320 : LREAL;
      AI_Tok_vozbuzhdeniia_vozbuditelia_LL AT %QL0.321 : LREAL;
      AI_Tok_vozbuzhdeniia_vozbuditelia_command AT %QW0.319 : UINT;
      AI_Tok_vozbuzhdeniia_vozbuditelia_newHL AT %QL0.322 : LREAL;
      AI_Tok_vozbuzhdeniia_vozbuditelia_newLL AT %QL0.323 : LREAL;
      AI_Tok_vozbuzhdeniia_vozbuditelia_status AT %QD0.324 : UDINT;
      AI_Tok_vozbuzhdeniia_vozbuditelia_value AT %QL0.325 : LREAL;
      AI_Uroven_masla_v_maslobake_HL AT %QL0.327 : LREAL;
      AI_Uroven_masla_v_maslobake_HW AT %QL0.328 : LREAL;
      AI_Uroven_masla_v_maslobake_LA AT %QL0.329 : LREAL;
      AI_Uroven_masla_v_maslobake_LL AT %QL0.330 : LREAL;
      AI_Uroven_masla_v_maslobake_LW AT %QL0.331 : LREAL;
      AI_Uroven_masla_v_maslobake_command AT %QW0.326 : UINT;
      AI_Uroven_masla_v_maslobake_newHL AT %QL0.332 : LREAL;
      AI_Uroven_masla_v_maslobake_newHW AT %QL0.333 : LREAL;
      AI_Uroven_masla_v_maslobake_newLA AT %QL0.334 : LREAL;
      AI_Uroven_masla_v_maslobake_newLL AT %QL0.335 : LREAL;
      AI_Uroven_masla_v_maslobake_newLW AT %QL0.336 : LREAL;
      AI_Uroven_masla_v_maslobake_status AT %QD0.337 : UDINT;
      AI_Uroven_masla_v_maslobake_value AT %QL0.338 : LREAL;
      AI_Vibratciia_STD_t1_HA AT %QL0.384 : LREAL;
      AI_Vibratciia_STD_t1_HL AT %QL0.385 : LREAL;
      AI_Vibratciia_STD_t1_HW AT %QL0.386 : LREAL;
      AI_Vibratciia_STD_t1_LL AT %QL0.387 : LREAL;
      AI_Vibratciia_STD_t1_command AT %QW0.383 : UINT;
      AI_Vibratciia_STD_t1_newHA AT %QL0.388 : LREAL;
      AI_Vibratciia_STD_t1_newHL AT %QL0.389 : LREAL;
      AI_Vibratciia_STD_t1_newHW AT %QL0.390 : LREAL;
      AI_Vibratciia_STD_t1_newLL AT %QL0.391 : LREAL;
      AI_Vibratciia_STD_t1_status AT %QD0.392 : UDINT;
      AI_Vibratciia_STD_t1_value AT %QL0.393 : LREAL;
      AI_Vibratciia_STD_t2_HA AT %QL0.395 : LREAL;
      AI_Vibratciia_STD_t2_HL AT %QL0.396 : LREAL;
      AI_Vibratciia_STD_t2_HW AT %QL0.397 : LREAL;
      AI_Vibratciia_STD_t2_LL AT %QL0.398 : LREAL;
      AI_Vibratciia_STD_t2_command AT %QW0.394 : UINT;
      AI_Vibratciia_STD_t2_newHA AT %QL0.399 : LREAL;
      AI_Vibratciia_STD_t2_newHL AT %QL0.400 : LREAL;
      AI_Vibratciia_STD_t2_newHW AT %QL0.401 : LREAL;
      AI_Vibratciia_STD_t2_newLL AT %QL0.402 : LREAL;
      AI_Vibratciia_STD_t2_status AT %QD0.403 : UDINT;
      AI_Vibratciia_STD_t2_value AT %QL0.404 : LREAL;
      AI_Vibratciia_rotora_nagnetatelia_t1_HA AT %QL0.340 : LREAL;
      AI_Vibratciia_rotora_nagnetatelia_t1_HL AT %QL0.341 : LREAL;
      AI_Vibratciia_rotora_nagnetatelia_t1_HW AT %QL0.342 : LREAL;
      AI_Vibratciia_rotora_nagnetatelia_t1_LL AT %QL0.343 : LREAL;
      AI_Vibratciia_rotora_nagnetatelia_t1_command AT %QW0.339 : UINT;
      AI_Vibratciia_rotora_nagnetatelia_t1_newHA AT %QL0.344 : LREAL;
      AI_Vibratciia_rotora_nagnetatelia_t1_newHL AT %QL0.345 : LREAL;
      AI_Vibratciia_rotora_nagnetatelia_t1_newHW AT %QL0.346 : LREAL;
      AI_Vibratciia_rotora_nagnetatelia_t1_newLL AT %QL0.347 : LREAL;
      AI_Vibratciia_rotora_nagnetatelia_t1_status AT %QD0.348 : UDINT;
      AI_Vibratciia_rotora_nagnetatelia_t1_value AT %QL0.349 : LREAL;
      AI_Vibratciia_rotora_nagnetatelia_t2_HA AT %QL0.351 : LREAL;
      AI_Vibratciia_rotora_nagnetatelia_t2_HL AT %QL0.352 : LREAL;
      AI_Vibratciia_rotora_nagnetatelia_t2_HW AT %QL0.353 : LREAL;
      AI_Vibratciia_rotora_nagnetatelia_t2_LL AT %QL0.354 : LREAL;
      AI_Vibratciia_rotora_nagnetatelia_t2_command AT %QW0.350 : UINT;
      AI_Vibratciia_rotora_nagnetatelia_t2_newHA AT %QL0.355 : LREAL;
      AI_Vibratciia_rotora_nagnetatelia_t2_newHL AT %QL0.356 : LREAL;
      AI_Vibratciia_rotora_nagnetatelia_t2_newHW AT %QL0.357 : LREAL;
      AI_Vibratciia_rotora_nagnetatelia_t2_newLL AT %QL0.358 : LREAL;
      AI_Vibratciia_rotora_nagnetatelia_t2_status AT %QD0.359 : UDINT;
      AI_Vibratciia_rotora_nagnetatelia_t2_value AT %QL0.360 : LREAL;
      AI_Vibratciia_rotora_nagnetatelia_t3_HA AT %QL0.362 : LREAL;
      AI_Vibratciia_rotora_nagnetatelia_t3_HL AT %QL0.363 : LREAL;
      AI_Vibratciia_rotora_nagnetatelia_t3_HW AT %QL0.364 : LREAL;
      AI_Vibratciia_rotora_nagnetatelia_t3_LL AT %QL0.365 : LREAL;
      AI_Vibratciia_rotora_nagnetatelia_t3_command AT %QW0.361 : UINT;
      AI_Vibratciia_rotora_nagnetatelia_t3_newHA AT %QL0.366 : LREAL;
      AI_Vibratciia_rotora_nagnetatelia_t3_newHL AT %QL0.367 : LREAL;
      AI_Vibratciia_rotora_nagnetatelia_t3_newHW AT %QL0.368 : LREAL;
      AI_Vibratciia_rotora_nagnetatelia_t3_newLL AT %QL0.369 : LREAL;
      AI_Vibratciia_rotora_nagnetatelia_t3_status AT %QD0.370 : UDINT;
      AI_Vibratciia_rotora_nagnetatelia_t3_value AT %QL0.371 : LREAL;
      AI_Vibratciia_rotora_nagnetatelia_t4_HA AT %QL0.373 : LREAL;
      AI_Vibratciia_rotora_nagnetatelia_t4_HL AT %QL0.374 : LREAL;
      AI_Vibratciia_rotora_nagnetatelia_t4_HW AT %QL0.375 : LREAL;
      AI_Vibratciia_rotora_nagnetatelia_t4_LL AT %QL0.376 : LREAL;
      AI_Vibratciia_rotora_nagnetatelia_t4_command AT %QW0.372 : UINT;
      AI_Vibratciia_rotora_nagnetatelia_t4_newHA AT %QL0.377 : LREAL;
      AI_Vibratciia_rotora_nagnetatelia_t4_newHL AT %QL0.378 : LREAL;
      AI_Vibratciia_rotora_nagnetatelia_t4_newHW AT %QL0.379 : LREAL;
      AI_Vibratciia_rotora_nagnetatelia_t4_newLL AT %QL0.380 : LREAL;
      AI_Vibratciia_rotora_nagnetatelia_t4_status AT %QD0.381 : UDINT;
      AI_Vibratciia_rotora_nagnetatelia_t4_value AT %QL0.382 : LREAL;
      AI_VoltageSHU_osnovnoi_vvod_HL AT %QL0.406 : LREAL;
      AI_VoltageSHU_osnovnoi_vvod_HW AT %QL0.407 : LREAL;
      AI_VoltageSHU_osnovnoi_vvod_LL AT %QL0.408 : LREAL;
      AI_VoltageSHU_osnovnoi_vvod_LW AT %QL0.409 : LREAL;
      AI_VoltageSHU_osnovnoi_vvod_command AT %QW0.405 : UINT;
      AI_VoltageSHU_osnovnoi_vvod_newHL AT %QL0.410 : LREAL;
      AI_VoltageSHU_osnovnoi_vvod_newHW AT %QL0.411 : LREAL;
      AI_VoltageSHU_osnovnoi_vvod_newLL AT %QL0.412 : LREAL;
      AI_VoltageSHU_osnovnoi_vvod_newLW AT %QL0.413 : LREAL;
      AI_VoltageSHU_osnovnoi_vvod_status AT %QD0.414 : UDINT;
      AI_VoltageSHU_osnovnoi_vvod_value AT %QL0.415 : LREAL;
      AI_VoltageSHU_rezervnyi_vvod_HL AT %QL0.417 : LREAL;
      AI_VoltageSHU_rezervnyi_vvod_HW AT %QL0.418 : LREAL;
      AI_VoltageSHU_rezervnyi_vvod_LL AT %QL0.419 : LREAL;
      AI_VoltageSHU_rezervnyi_vvod_LW AT %QL0.420 : LREAL;
      AI_VoltageSHU_rezervnyi_vvod_command AT %QW0.416 : UINT;
      AI_VoltageSHU_rezervnyi_vvod_newHL AT %QL0.421 : LREAL;
      AI_VoltageSHU_rezervnyi_vvod_newHW AT %QL0.422 : LREAL;
      AI_VoltageSHU_rezervnyi_vvod_newLL AT %QL0.423 : LREAL;
      AI_VoltageSHU_rezervnyi_vvod_newLW AT %QL0.424 : LREAL;
      AI_VoltageSHU_rezervnyi_vvod_status AT %QD0.425 : UDINT;
      AI_VoltageSHU_rezervnyi_vvod_value AT %QL0.426 : LREAL;
      AI_dP_gaza_na_konfuzore_nagnetatelia_HL AT %QL0.9 : LREAL;
      AI_dP_gaza_na_konfuzore_nagnetatelia_LL AT %QL0.10 : LREAL;
      AI_dP_gaza_na_konfuzore_nagnetatelia_command AT %QW0.8 : UINT;
      AI_dP_gaza_na_konfuzore_nagnetatelia_newHL AT %QL0.11 : LREAL;
      AI_dP_gaza_na_konfuzore_nagnetatelia_newLL AT %QL0.12 : LREAL;
      AI_dP_gaza_na_konfuzore_nagnetatelia_status AT %QD0.13 : UDINT;
      AI_dP_gaza_na_konfuzore_nagnetatelia_value AT %QL0.14 : LREAL;
      AI_dPmaslo_gaz_HL AT %QL0.16 : LREAL;
      AI_dPmaslo_gaz_LA AT %QL0.17 : LREAL;
      AI_dPmaslo_gaz_LL AT %QL0.18 : LREAL;
      AI_dPmaslo_gaz_LW AT %QL0.19 : LREAL;
      AI_dPmaslo_gaz_MaxChangeDown AT %QL0.877 : LREAL;
      AI_dPmaslo_gaz_MaxChangeUP AT %QL0.876 : LREAL;
      AI_dPmaslo_gaz_command AT %QW0.15 : UINT;
      AI_dPmaslo_gaz_newHL AT %QL0.20 : LREAL;
      AI_dPmaslo_gaz_newLA AT %QL0.21 : LREAL;
      AI_dPmaslo_gaz_newLL AT %QL0.22 : LREAL;
      AI_dPmaslo_gaz_newLW AT %QL0.23 : LREAL;
      AI_dPmaslo_gaz_newMaxChangeDown AT %QL0.875 : LREAL;
      AI_dPmaslo_gaz_newMaxChangeUP AT %QL0.874 : LREAL;
      AI_dPmaslo_gaz_status AT %QD0.24 : UDINT;
      AI_dPmaslo_gaz_value AT %QL0.25 : LREAL;
      A1_10_err_mode AT %QW0.825 : UINT;
      A1_11_err_mode AT %QW0.826 : UINT;
      A1_12_err_mode AT %QW0.827 : UINT;
      A1_13_err_mode AT %QW0.828 : UINT;
      A1_14_err_mode AT %QW0.829 : UINT;
      A1_15_err_mode AT %QW0.830 : UINT;
      A1_1_err_mode AT %QW0.816 : UINT;
      A1_2_err_mode AT %QW0.817 : UINT;
      A1_3_err_mode AT %QW0.818 : UINT;
      A1_4_err_mode AT %QW0.819 : UINT;
      A1_5_err_mode AT %QW0.820 : UINT;
      A1_6_err_mode AT %QW0.821 : UINT;
      A1_7_err_mode AT %QW0.822 : UINT;
      A1_8_err_mode AT %QW0.823 : UINT;
      A1_9_err_mode AT %QW0.824 : UINT;
      A2_10_err_mode AT %QW0.840 : UINT;
      A2_11_err_mode AT %QW0.841 : UINT;
      A2_12_err_mode AT %QW0.842 : UINT;
      A2_13_err_mode AT %QW0.843 : UINT;
      A2_14_err_mode AT %QW0.844 : UINT;
      A2_15_err_mode AT %QW0.845 : UINT;
      A2_1_err_mode AT %QW0.831 : UINT;
      A2_2_err_mode AT %QW0.832 : UINT;
      A2_3_err_mode AT %QW0.833 : UINT;
      A2_4_err_mode AT %QW0.834 : UINT;
      A2_5_err_mode AT %QW0.835 : UINT;
      A2_6_err_mode AT %QW0.836 : UINT;
      A2_7_err_mode AT %QW0.837 : UINT;
      A2_8_err_mode AT %QW0.838 : UINT;
      A2_9_err_mode AT %QW0.839 : UINT;
      AI_0_dblValue AT %QL0.736 : LREAL;
      AI_10_dblValue AT %QL0.746 : LREAL;
      AI_11_dblValue AT %QL0.747 : LREAL;
      AI_12_dblValue AT %QL0.748 : LREAL;
      AI_13_dblValue AT %QL0.749 : LREAL;
      AI_14_dblValue AT %QL0.750 : LREAL;
      AI_15_dblValue AT %QL0.751 : LREAL;
      AI_16_dblValue AT %QL0.752 : LREAL;
      AI_17_dblValue AT %QL0.753 : LREAL;
      AI_18_dblValue AT %QL0.754 : LREAL;
      AI_19_dblValue AT %QL0.755 : LREAL;
      AI_1_dblValue AT %QL0.737 : LREAL;
      AI_20_dblValue AT %QL0.756 : LREAL;
      AI_21_dblValue AT %QL0.757 : LREAL;
      AI_22_dblValue AT %QL0.758 : LREAL;
      AI_23_dblValue AT %QL0.759 : LREAL;
      AI_24_dblValue AT %QL0.760 : LREAL;
      AI_25_dblValue AT %QL0.761 : LREAL;
      AI_26_dblValue AT %QL0.762 : LREAL;
      AI_27_dblValue AT %QL0.763 : LREAL;
      AI_28_dblValue AT %QL0.764 : LREAL;
      AI_29_dblValue AT %QL0.765 : LREAL;
      AI_2_dblValue AT %QL0.738 : LREAL;
      AI_30_dblValue AT %QL0.766 : LREAL;
      AI_31_dblValue AT %QL0.767 : LREAL;
      AI_32_dblValue AT %QL0.768 : LREAL;
      AI_33_dblValue AT %QL0.769 : LREAL;
      AI_34_dblValue AT %QL0.770 : LREAL;
      AI_35_dblValue AT %QL0.771 : LREAL;
      AI_36_dblValue AT %QL0.772 : LREAL;
      AI_37_dblValue AT %QL0.773 : LREAL;
      AI_38_dblValue AT %QL0.774 : LREAL;
      AI_39_dblValue AT %QL0.775 : LREAL;
      AI_3_dblValue AT %QL0.739 : LREAL;
      AI_40_dblValue AT %QL0.776 : LREAL;
      AI_41_dblValue AT %QL0.777 : LREAL;
      AI_42_dblValue AT %QL0.778 : LREAL;
      AI_43_dblValue AT %QL0.779 : LREAL;
      AI_44_dblValue AT %QL0.780 : LREAL;
      AI_45_dblValue AT %QL0.781 : LREAL;
      AI_46_dblValue AT %QL0.782 : LREAL;
      AI_47_dblValue AT %QL0.783 : LREAL;
      AI_48_dblValue AT %QL0.784 : LREAL;
      AI_49_dblValue AT %QL0.785 : LREAL;
      AI_4_dblValue AT %QL0.740 : LREAL;
      AI_50_dblValue AT %QL0.786 : LREAL;
      AI_51_dblValue AT %QL0.787 : LREAL;
      AI_52_dblValue AT %QL0.788 : LREAL;
      AI_53_dblValue AT %QL0.789 : LREAL;
      AI_54_dblValue AT %QL0.790 : LREAL;
      AI_55_dblValue AT %QL0.791 : LREAL;
      AI_56_dblValue AT %QL0.792 : LREAL;
      AI_57_dblValue AT %QL0.793 : LREAL;
      AI_58_dblValue AT %QL0.794 : LREAL;
      AI_59_dblValue AT %QL0.795 : LREAL;
      AI_5_dblValue AT %QL0.741 : LREAL;
      AI_60_dblValue AT %QL0.796 : LREAL;
      AI_61_dblValue AT %QL0.797 : LREAL;
      AI_62_dblValue AT %QL0.798 : LREAL;
      AI_63_dblValue AT %QL0.799 : LREAL;
      AI_64_dblValue AT %QL0.800 : LREAL;
      AI_65_dblValue AT %QL0.801 : LREAL;
      AI_66_dblValue AT %QL0.802 : LREAL;
      AI_67_dblValue AT %QL0.803 : LREAL;
      AI_68_dblValue AT %QL0.804 : LREAL;
      AI_69_dblValue AT %QL0.805 : LREAL;
      AI_6_dblValue AT %QL0.742 : LREAL;
      AI_70_dblValue AT %QL0.806 : LREAL;
      AI_71_dblValue AT %QL0.807 : LREAL;
      AI_72_dblValue AT %QL0.808 : LREAL;
      AI_73_dblValue AT %QL0.809 : LREAL;
      AI_74_dblValue AT %QL0.810 : LREAL;
      AI_75_dblValue AT %QL0.811 : LREAL;
      AI_76_dblValue AT %QL0.812 : LREAL;
      AI_77_dblValue AT %QL0.813 : LREAL;
      AI_78_dblValue AT %QL0.814 : LREAL;
      AI_79_dblValue AT %QL0.815 : LREAL;
      AI_7_dblValue AT %QL0.743 : LREAL;
      AI_8_dblValue AT %QL0.744 : LREAL;
      AI_9_dblValue AT %QL0.745 : LREAL;
      BS_Core1 AT %QD0.603 : REAL;
      BS_Core2 AT %QD0.675 : REAL;
      BS_Core3 AT %QD0.683 : REAL;
      BS_Core4 AT %QD0.709 : REAL;
      BS_FreeMemory AT %QD0.730 : REAL;
      BS_Temp1 AT %QD0.734 : REAL;
      BS_Temp2 AT %QD0.735 : REAL;
      DI_0_1_wValue AT %QD0.852 : UDINT;
      DI_10_11_wValue AT %QD0.857 : UDINT;
      DI_12_13_wValue AT %QD0.858 : UDINT;
      DI_14_15_wValue AT %QD0.859 : UDINT;
      DI_16_17_wValue AT %QD0.860 : UDINT;
      DI_18_19_wValue AT %QD0.861 : UDINT;
      DI_20_21_wValue AT %QD0.862 : UDINT;
      DI_2_3_wValue AT %QD0.853 : UDINT;
      DI_4_5_wValue AT %QD0.854 : UDINT;
      DI_6_7_wValue AT %QD0.855 : UDINT;
      DI_8_9_wValue AT %QD0.856 : UDINT;
      DO_0_wValue AT %QW0.846 : UINT;
      DO_1_wValue AT %QW0.847 : UINT;
      DO_2_wValue AT %QW0.848 : UINT;
      DO_3_wValue AT %QW0.849 : UINT;
      DO_4_wValue AT %QW0.850 : UINT;
      DO_5_wValue AT %QW0.851 : UINT;
      IM_SingleSignals_DverShkafaOtkryta_status AT %QD0.456 : UDINT;
      IM_SingleSignals_KZ_10kv_status AT %QD0.457 : UDINT;
      IM_SingleSignals_NOGPA_knopkaSHU_status AT %QD0.453 : UDINT;
      IM_SingleSignals_NS_G10_G11_status AT %QD0.481 : UDINT;
      IM_SingleSignals_NS_G13_G14_status AT %QD0.482 : UDINT;
      IM_SingleSignals_NS_G15_G16_status AT %QD0.483 : UDINT;
      IM_SingleSignals_NS_G17_status AT %QD0.484 : UDINT;
      IM_SingleSignals_NS_G18_G19_status AT %QD0.485 : UDINT;
      IM_SingleSignals_NS_G1_G2_status AT %QD0.477 : UDINT;
      IM_SingleSignals_NS_G3_G4_status AT %QD0.478 : UDINT;
      IM_SingleSignals_NS_G5_G6_status AT %QD0.479 : UDINT;
      IM_SingleSignals_NS_G7_G8_status AT %QD0.480 : UDINT;
      IM_SingleSignals_OsevoiSdvig_levo_status AT %QD0.458 : UDINT;
      IM_SingleSignals_OsevoiSdvig_pravo_status AT %QD0.459 : UDINT;
      IM_SingleSignals_P_oil_low_status AT %QD0.455 : UDINT;
      IM_SingleSignals_QF10_QF11_on_status AT %QD0.463 : UDINT;
      IM_SingleSignals_QF12_QF13_on_status AT %QD0.464 : UDINT;
      IM_SingleSignals_QF14_QF15_on_status AT %QD0.465 : UDINT;
      IM_SingleSignals_QF1_on_status AT %QD0.466 : UDINT;
      IM_SingleSignals_QF22_on_status AT %QD0.476 : UDINT;
      IM_SingleSignals_QF23_on_status AT %QD0.468 : UDINT;
      IM_SingleSignals_QF2_on_status AT %QD0.467 : UDINT;
      IM_SingleSignals_QF4_QF5_on_status AT %QD0.460 : UDINT;
      IM_SingleSignals_QF6_QF7_on_status AT %QD0.461 : UDINT;
      IM_SingleSignals_QF8_QF9_on_status AT %QD0.462 : UDINT;
      IM_SingleSignals_Vozb_AsinchHod_status AT %QD0.469 : UDINT;
      IM_SingleSignals_Vozb_ControlVozbuditela_status AT %QD0.470 : UDINT;
      IM_SingleSignals_Vozb_KontaktorON_status AT %QD0.471 : UDINT;
      IM_SingleSignals_Vozb_Overload_status AT %QD0.472 : UDINT;
      IM_SingleSignals_Vozb_ProboiVentila_status AT %QD0.473 : UDINT;
      IM_SingleSignals_Vozb_ReSynchronize_status AT %QD0.474 : UDINT;
      IM_SingleSignals_dP_gazgaz_Kran1_status AT %QD0.454 : UDINT;
      IM_SingleSignals_dP_oilgaz_low_status AT %QD0.475 : UDINT;
      IM_Ten_inCommand_ARM AT %QW0.447 : UINT;
      IM_Ten_status AT %QD0.448 : UDINT;
      IM_kran1_inCommand_ARM AT %QW0.427 : UINT;
      IM_kran1_status AT %QD0.428 : UDINT;
      IM_kran2_inCommand_ARM AT %QW0.429 : UINT;
      IM_kran2_status AT %QD0.430 : UDINT;
      IM_kran3b_inCommand_ARM AT %QW0.431 : UINT;
      IM_kran3b_status AT %QD0.432 : UDINT;
      IM_kran4_inCommand_ARM AT %QW0.433 : UINT;
      IM_kran4_status AT %QD0.434 : UDINT;
      IM_kran5_inCommand_ARM AT %QW0.435 : UINT;
      IM_kran5_status AT %QD0.436 : UDINT;
      IM_kran6_inCommand_ARM AT %QW0.437 : UINT;
      IM_kran6_status AT %QD0.438 : UDINT;
      IM_mv_inCommand_ARM AT %QW0.439 : UINT;
      IM_mv_status AT %QD0.440 : UDINT;
      IM_nu1_inCommand_ARM AT %QW0.441 : UINT;
      IM_nu1_status AT %QD0.442 : UDINT;
      IM_nu2_inCommand_ARM AT %QW0.443 : UINT;
      IM_nu2_status AT %QD0.444 : UDINT;
      IM_pns_inCommand_ARM AT %QW0.445 : UINT;
      IM_pns_status AT %QD0.446 : UDINT;
      IM_v1_Avom_inCommand_ARM AT %QW0.449 : UINT;
      IM_v1_Avom_status AT %QD0.450 : UDINT;
      IM_v2_Avom_inCommand_ARM AT %QW0.451 : UINT;
      IM_v2_Avom_status AT %QD0.452 : UDINT;
      algManager_Mode AT %QW0.732 : UINT;
      algoritms_AntiPompag_UgolVNA_Value AT %QL0.726 : LREAL;
      algoritms_AntiPompag_UgolVNA_inCommand_ARM AT %QW0.605 : UINT;
      algoritms_AntiPompag_UgolVNA_newValue AT %QL0.606 : LREAL;
      algoritms_AntiPompag_UgolVNA_status AT %QD0.725 : UDINT;
      algoritms_AntiPompag_q_Value AT %QL0.724 : LREAL;
      algoritms_AntiPompag_q_inCommand_ARM AT %QW0.604 : UINT;
      algoritms_AntiPompag_q_status AT %QD0.723 : UDINT;
      algoritms_AntiPompag_zapas_Value AT %QL0.728 : LREAL;
      algoritms_AntiPompag_zapas_inCommand_ARM AT %QW0.607 : UINT;
      algoritms_AntiPompag_zapas_status AT %QD0.727 : UDINT;
      algoritms_Apusk_Error AT %QD0.689 : UDINT;
      algoritms_Apusk_Start AT %QD0.688 : UDINT;
      algoritms_Apusk_Top AT %QD0.690 : UDINT;
      algoritms_Apusk_inCommand_ARM AT %QW0.555 : UINT;
      algoritms_Apusk_status AT %QD0.687 : UDINT;
      algoritms_AutoAvom_hysteresis_Value AT %QL0.716 : LREAL;
      algoritms_AutoAvom_hysteresis_inCommand_ARM AT %QW0.556 : UINT;
      algoritms_AutoAvom_hysteresis_newValue AT %QL0.557 : LREAL;
      algoritms_AutoAvom_hysteresis_status AT %QD0.715 : UDINT;
      algoritms_AutoAvom_inCommand_ARM AT %QW0.562 : UINT;
      algoritms_AutoAvom_on1Temperature_Value AT %QL0.712 : LREAL;
      algoritms_AutoAvom_on1Temperature_inCommand_ARM AT %QW0.558 : UINT;
      algoritms_AutoAvom_on1Temperature_newValue AT %QL0.559 : LREAL;
      algoritms_AutoAvom_on1Temperature_status AT %QD0.711 : UDINT;
      algoritms_AutoAvom_on2Temperature_Value AT %QL0.714 : LREAL;
      algoritms_AutoAvom_on2Temperature_inCommand_ARM AT %QW0.560 : UINT;
      algoritms_AutoAvom_on2Temperature_newValue AT %QL0.561 : LREAL;
      algoritms_AutoAvom_on2Temperature_status AT %QD0.713 : UDINT;
      algoritms_AutoAvom_status AT %QD0.710 : UDINT;
      algoritms_AutoPns_OffTimer AT %QW0.701 : UINT;
      algoritms_AutoPns_OnTimer AT %QW0.700 : UINT;
      algoritms_AutoPns_Ust_Run_Value AT %QL0.703 : LREAL;
      algoritms_AutoPns_Ust_Run_inCommand_ARM AT %QW0.567 : UINT;
      algoritms_AutoPns_Ust_Run_newValue AT %QL0.568 : LREAL;
      algoritms_AutoPns_Ust_Run_status AT %QD0.702 : UDINT;
      algoritms_AutoPns_Ust_Stop_Value AT %QL0.705 : LREAL;
      algoritms_AutoPns_Ust_Stop_inCommand_ARM AT %QW0.569 : UINT;
      algoritms_AutoPns_Ust_Stop_newValue AT %QL0.570 : LREAL;
      algoritms_AutoPns_Ust_Stop_status AT %QD0.704 : UDINT;
      algoritms_AutoPns_inCommand_ARM AT %QW0.571 : UINT;
      algoritms_AutoPns_status AT %QD0.699 : UDINT;
      algoritms_AutoTen_inCommand_ARM AT %QW0.610 : UINT;
      algoritms_AutoTen_offTemperature_Value AT %QL0.721 : LREAL;
      algoritms_AutoTen_offTemperature_inCommand_ARM AT %QW0.608 : UINT;
      algoritms_AutoTen_offTemperature_newValue AT %QL0.609 : LREAL;
      algoritms_AutoTen_offTemperature_status AT %QD0.720 : UDINT;
      algoritms_AutoTen_status AT %QD0.719 : UDINT;
      algoritms_Remont_inCommand_ARM AT %QW0.585 : UINT;
      algoritms_Remont_status AT %QD0.718 : UDINT;
      algoritms_RingToLine_Error AT %QD0.667 : UDINT;
      algoritms_RingToLine_Start AT %QD0.666 : UDINT;
      algoritms_RingToLine_Top AT %QD0.668 : UDINT;
      algoritms_RingToLine_inCommand_ARM AT %QW0.586 : UINT;
      algoritms_RingToLine_status AT %QD0.665 : UDINT;
      algoritms_SemiAutoPusk_Error AT %QD0.693 : UDINT;
      algoritms_SemiAutoPusk_Start AT %QD0.692 : UDINT;
      algoritms_SemiAutoPusk_Top AT %QD0.694 : UDINT;
      algoritms_SemiAutoPusk_cmdRun1ph_inCommand_ARM AT %QW0.587 : UINT;
      algoritms_SemiAutoPusk_cmdRun1ph_status AT %QD0.695 : UDINT;
      algoritms_SemiAutoPusk_cmdRun2ph_inCommand_ARM AT %QW0.588 : UINT;
      algoritms_SemiAutoPusk_cmdRun2ph_status AT %QD0.696 : UDINT;
      algoritms_SemiAutoPusk_cmdRun3ph_inCommand_ARM AT %QW0.589 : UINT;
      algoritms_SemiAutoPusk_cmdRun3ph_status AT %QD0.697 : UDINT;
      algoritms_SemiAutoPusk_cmdRun4ph_inCommand_ARM AT %QW0.590 : UINT;
      algoritms_SemiAutoPusk_cmdRun4ph_status AT %QD0.698 : UDINT;
      algoritms_SemiAutoPusk_inCommand_ARM AT %QW0.591 : UINT;
      algoritms_SemiAutoPusk_status AT %QD0.691 : UDINT;
      algoritms_TestProtection_inCommand_ARM AT %QW0.600 : UINT;
      algoritms_TestProtection_status AT %QD0.717 : UDINT;
      algoritms_ao_Error AT %QD0.617 : UDINT;
      algoritms_ao_Start AT %QD0.616 : UDINT;
      algoritms_ao_Top AT %QD0.618 : UDINT;
      algoritms_ao_inCommand_ARM AT %QW0.554 : UINT;
      algoritms_ao_status AT %QD0.619 : UDINT;
      algoritms_ao_waitKran_timer AT %QW0.620 : UINT;
      algoritms_autoNu_NotHasRezervNU AT %QX0.729 : BOOL;
      algoritms_autoNu_Reset_HasNU AT %QX0.731 : BOOL;
      algoritms_autoNu_Ust_Swap_Value AT %QL0.708 : LREAL;
      algoritms_autoNu_Ust_Swap_inCommand_ARM AT %QW0.563 : UINT;
      algoritms_autoNu_Ust_Swap_newValue AT %QL0.564 : LREAL;
      algoritms_autoNu_Ust_Swap_status AT %QD0.707 : UDINT;
      algoritms_autoNu_inCommand_ARM AT %QW0.566 : UINT;
      algoritms_autoNu_mainNU_inCommand_ARM AT %QW0.565 : UINT;
      algoritms_autoNu_mainNU_status AT %QD0.722 : UDINT;
      algoritms_autoNu_status AT %QD0.706 : UDINT;
      algoritms_engineRun_BreakPuskTimer_timer AT %QW0.657 : UINT;
      algoritms_engineRun_Error AT %QD0.655 : UDINT;
      algoritms_engineRun_Start AT %QD0.654 : UDINT;
      algoritms_engineRun_Top AT %QD0.656 : UDINT;
      algoritms_engineRun_inCommand_ARM AT %QW0.572 : UINT;
      algoritms_engineRun_status AT %QD0.653 : UDINT;
      algoritms_filling_BreakPuskTimer_timer AT %QW0.662 : UINT;
      algoritms_filling_Error AT %QD0.660 : UDINT;
      algoritms_filling_Start AT %QD0.659 : UDINT;
      algoritms_filling_Top AT %QD0.661 : UDINT;
      algoritms_filling_inCommand_ARM AT %QW0.573 : UINT;
      algoritms_filling_status AT %QD0.658 : UDINT;
      algoritms_filling_waitAfterKran4_timer AT %QW0.663 : UINT;
      algoritms_filling_waitAfterKran5_timer AT %QW0.664 : UINT;
      algoritms_no_Error AT %QD0.612 : UDINT;
      algoritms_no_Start AT %QD0.611 : UDINT;
      algoritms_no_Top AT %QD0.613 : UDINT;
      algoritms_no_inCommand_ARM AT %QW0.574 : UINT;
      algoritms_no_status AT %QD0.614 : UDINT;
      algoritms_no_waitCloseKran_timer AT %QW0.615 : UINT;
      algoritms_ppu_Error AT %QD0.643 : UDINT;
      algoritms_ppu_Start AT %QD0.642 : UDINT;
      algoritms_ppu_Top AT %QD0.644 : UDINT;
      algoritms_ppu_inCommand_ARM AT %QW0.575 : UINT;
      algoritms_ppu_status AT %QD0.641 : UDINT;
      algoritms_puskK_Error AT %QD0.673 : UDINT;
      algoritms_puskK_Start AT %QD0.672 : UDINT;
      algoritms_puskK_Top AT %QD0.674 : UDINT;
      algoritms_puskK_inCommand_ARM AT %QW0.578 : UINT;
      algoritms_puskK_questionFilling_inCommand_ARM AT %QW0.576 : UINT;
      algoritms_puskK_questionFilling_status AT %QD0.677 : UDINT;
      algoritms_puskK_questionUnload_inCommand_ARM AT %QW0.577 : UINT;
      algoritms_puskK_questionUnload_status AT %QD0.678 : UDINT;
      algoritms_puskK_status AT %QD0.671 : UDINT;
      algoritms_puskK_wait720_timer AT %QW0.676 : UINT;
      algoritms_puskOilSystem_BreakPuskTimer_Poil_timer AT %QW0.649 : UINT;
      algoritms_puskOilSystem_BreakPuskTimer_dPmg_timer AT %QW0.650 : UINT;
      algoritms_puskOilSystem_Error AT %QD0.647 : UDINT;
      algoritms_puskOilSystem_Start AT %QD0.646 : UDINT;
      algoritms_puskOilSystem_Top AT %QD0.648 : UDINT;
      algoritms_puskOilSystem_Ust_dPmg_Value AT %QL0.652 : LREAL;
      algoritms_puskOilSystem_Ust_dPmg_inCommand_ARM AT %QW0.579 : UINT;
      algoritms_puskOilSystem_Ust_dPmg_newValue AT %QL0.580 : LREAL;
      algoritms_puskOilSystem_Ust_dPmg_status AT %QD0.651 : UDINT;
      algoritms_puskOilSystem_inCommand_ARM AT %QW0.581 : UINT;
      algoritms_puskOilSystem_status AT %QD0.645 : UDINT;
      algoritms_puskV_Error AT %QD0.681 : UDINT;
      algoritms_puskV_Start AT %QD0.680 : UDINT;
      algoritms_puskV_Top AT %QD0.682 : UDINT;
      algoritms_puskV_inCommand_ARM AT %QW0.584 : UINT;
      algoritms_puskV_questionFilling_inCommand_ARM AT %QW0.582 : UINT;
      algoritms_puskV_questionFilling_status AT %QD0.685 : UDINT;
      algoritms_puskV_questionMVoff_inCommand_ARM AT %QW0.583 : UINT;
      algoritms_puskV_questionMVoff_status AT %QD0.686 : UDINT;
      algoritms_puskV_status AT %QD0.679 : UDINT;
      algoritms_puskV_wait600_timer AT %QW0.684 : UINT;
      algoritms_testIm_TypeSwitch_inCommand_ARM AT %QW0.596 : UINT;
      algoritms_testIm_TypeSwitch_status AT %QD0.640 : UDINT;
      algoritms_testIm_inCommand_ARM AT %QW0.597 : UINT;
      algoritms_testIm_status AT %QD0.639 : UDINT;
      algoritms_testPms_BreakTest_timer AT %QW0.631 : UINT;
      algoritms_testPms_Error AT %QD0.628 : UDINT;
      algoritms_testPms_Start AT %QD0.627 : UDINT;
      algoritms_testPms_Top AT %QD0.629 : UDINT;
      algoritms_testPms_algContinue_inCommand_ARM AT %QW0.598 : UINT;
      algoritms_testPms_algContinue_status AT %QD0.669 : UDINT;
      algoritms_testPms_inCommand_ARM AT %QW0.599 : UINT;
      algoritms_testPms_status AT %QD0.630 : UDINT;
      algoritms_testdPmg_BreakTest_timer AT %QW0.636 : UINT;
      algoritms_testdPmg_Error AT %QD0.633 : UDINT;
      algoritms_testdPmg_Start AT %QD0.632 : UDINT;
      algoritms_testdPmg_Top AT %QD0.634 : UDINT;
      algoritms_testdPmg_Ust_dPLow_Value AT %QL0.638 : LREAL;
      algoritms_testdPmg_Ust_dPLow_inCommand_ARM AT %QW0.593 : UINT;
      algoritms_testdPmg_Ust_dPLow_newValue AT %QL0.594 : LREAL;
      algoritms_testdPmg_Ust_dPLow_status AT %QD0.637 : UDINT;
      algoritms_testdPmg_algContinue_inCommand_ARM AT %QW0.592 : UINT;
      algoritms_testdPmg_algContinue_status AT %QD0.670 : UDINT;
      algoritms_testdPmg_inCommand_ARM AT %QW0.595 : UINT;
      algoritms_testdPmg_status AT %QD0.635 : UDINT;
      algoritms_vibegPNS_Error AT %QD0.622 : UDINT;
      algoritms_vibegPNS_Start AT %QD0.621 : UDINT;
      algoritms_vibegPNS_Top AT %QD0.623 : UDINT;
      algoritms_vibegPNS_algContinue_inCommand_ARM AT %QW0.601 : UINT;
      algoritms_vibegPNS_algContinue_status AT %QD0.626 : UDINT;
      algoritms_vibegPNS_inCommand_ARM AT %QW0.602 : UINT;
      algoritms_vibegPNS_status AT %QD0.624 : UDINT;
      algoritms_vibegPNS_waitVibeg_timer AT %QW0.625 : UINT;
      protectManager_protectionInRemont AT %QX0.733 : BOOL;
      protections_AOKC_SHKC_command AT %QW0.908 : UINT;
      protections_AOKC_SHKC_status AT %QW0.515 : UINT;
      protections_AO_PRU_command AT %QW0.909 : UINT;
      protections_AO_PRU_status AT %QW0.516 : UINT;
      protections_AO_ot_SHU_command AT %QW0.910 : UINT;
      protections_AO_ot_SHU_status AT %QW0.517 : UINT;
      protections_Fprotectionsl_chastotnii_pusk_command AT %QW0.906 : UINT;
      protections_Fprotectionsl_chastotnii_pusk_status AT %QW0.513 : UINT;
      protections_Kran1_sdvig_command AT %QW0.912 : UINT;
      protections_Kran1_sdvig_status AT %QW0.519 : UINT;
      protections_Kran2_sdvig_command AT %QW0.913 : UINT;
      protections_Kran2_sdvig_status AT %QW0.878 : UINT;
      protections_Off_avar_vikluchatel_command AT %QW0.907 : UINT;
      protections_Off_avar_vikluchatel_status AT %QW0.514 : UINT;
      protections_Os_sdvig_nagnetatelja_minus_command AT %QW0.891 : UINT;
      protections_Os_sdvig_nagnetatelja_minus_status AT %QW0.498 : UINT;
      protections_Os_sdvig_nagnetatelja_plus_command AT %QW0.890 : UINT;
      protections_Os_sdvig_nagnetatelja_plus_status AT %QW0.497 : UINT;
      protections_Pgaza_na_vhode_nagnetatelia_GPA_STOP_command AT %QW0.893 : UINT;
      protections_Pgaza_na_vhode_nagnetatelia_GPA_STOP_status AT %QW0.500 : UINT;
      protections_Pgaza_na_vyhode_nagnetatelia_GPA_STOP_command AT %QW0.892 : UINT;
      protections_Pgaza_na_vyhode_nagnetatelia_GPA_STOP_status AT %QW0.499 : UINT;
      protections_Pgaza_na_vyhode_nagnetatelia_command AT %QW0.894 : UINT;
      protections_Pgaza_na_vyhode_nagnetatelia_status AT %QW0.501 : UINT;
      protections_Pmaslo_sm_nizkoe_command AT %QW0.896 : UINT;
      protections_Pmaslo_sm_nizkoe_status AT %QW0.503 : UINT;
      protections_Pmaslo_sm_vysokoe_command AT %QW0.897 : UINT;
      protections_Pmaslo_sm_vysokoe_status AT %QW0.504 : UINT;
      protections_Reg_vozb_off_command AT %QW0.905 : UINT;
      protections_Reg_vozb_off_status AT %QW0.512 : UINT;
      protections_Tgaza_na_vyhode_H_command AT %QW0.889 : UINT;
      protections_Tgaza_na_vyhode_H_status AT %QW0.496 : UINT;
      protections_To_podshipnika_N_EDT_7_command AT %QW0.885 : UINT;
      protections_To_podshipnika_N_EDT_7_status AT %QW0.492 : UINT;
      protections_To_podshipnika_shest_red_EDT_5_command AT %QW0.883 : UINT;
      protections_To_podshipnika_shest_red_EDT_5_status AT %QW0.490 : UINT;
      protections_To_podshipnika_shest_red_EDT_6_command AT %QW0.884 : UINT;
      protections_To_podshipnika_shest_red_EDT_6_status AT %QW0.491 : UINT;
      protections_To_podshipnika_svob_konca_EDT_8_command AT %QW0.886 : UINT;
      protections_To_podshipnika_svob_konca_EDT_8_status AT %QW0.493 : UINT;
      protections_Topornogo_podshipnika_EDT_1_command AT %QW0.879 : UINT;
      protections_Topornogo_podshipnika_EDT_1_status AT %QW0.486 : UINT;
      protections_Toy_podshipnika_EDT_2_command AT %QW0.880 : UINT;
      protections_Toy_podshipnika_EDT_2_status AT %QW0.487 : UINT;
      protections_Toy_podshipnika_kol_EDT_3_command AT %QW0.881 : UINT;
      protections_Toy_podshipnika_kol_EDT_3_status AT %QW0.488 : UINT;
      protections_Toy_podshipnika_kol_EDT_4_command AT %QW0.882 : UINT;
      protections_Toy_podshipnika_kol_EDT_4_status AT %QW0.489 : UINT;
      protections_Ty_podshipnika_rab_kol_EDT_9_command AT %QW0.887 : UINT;
      protections_Ty_podshipnika_rab_kol_EDT_9_status AT %QW0.494 : UINT;
      protections_Typornogo_podshipnika_nerab_kolodok_HT_10_command AT %QW0.888 : UINT;
      protections_Typornogo_podshipnika_nerab_kolodok_HT_10_status AT %QW0.495 : UINT;
      protections_Vibro_skorost_OPED_T1_command AT %QW0.898 : UINT;
      protections_Vibro_skorost_OPED_T1_status AT %QW0.505 : UINT;
      protections_Vibro_skorost_OPED_T2_command AT %QW0.899 : UINT;
      protections_Vibro_skorost_OPED_T2_status AT %QW0.506 : UINT;
      protections_Vibro_skorost_OP_kolesa_RH_T4_command AT %QW0.901 : UINT;
      protections_Vibro_skorost_OP_kolesa_RH_T4_status AT %QW0.508 : UINT;
      protections_Vibro_skorost_OP_shesterni_RED_T5_command AT %QW0.902 : UINT;
      protections_Vibro_skorost_OP_shesterni_RED_T5_status AT %QW0.509 : UINT;
      protections_Vibro_skorost_OP_shesterni_RED_T6_command AT %QW0.903 : UINT;
      protections_Vibro_skorost_OP_shesterni_RED_T6_status AT %QW0.510 : UINT;
      protections_Vibro_skorost_OYP_kolesa_ED_T3_command AT %QW0.900 : UINT;
      protections_Vibro_skorost_OYP_kolesa_ED_T3_status AT %QW0.507 : UINT;
      protections_dPmaslo_gaz_command AT %QW0.895 : UINT;
      protections_dPmaslo_gaz_less100_command AT %QW0.904 : UINT;
      protections_dPmaslo_gaz_less100_status AT %QW0.511 : UINT;
      protections_dPmaslo_gaz_status AT %QW0.502 : UINT;
      protections_mvOff_command AT %QW0.911 : UINT;
      protections_mvOff_status AT %QW0.518 : UINT;
    END_VAR
    TASK task0(INTERVAL := T#20ms,PRIORITY := 0);
    PROGRAM instance0 WITH task0 : program0;
  END_RESOURCE
END_CONFIGURATION
